KUKA KRL program: AutoChangeToolSps.src, AutoChangeToolSps.dat

--- AutoChangeToolSps.src ---
&ACCESS RV
&REL 153
&COMMENT Ansteuerung Micromaster Frequenzumrichter
&PARAM EDITMASK = *
&PARAM TEMPLATE = C:\KRC\Roboter\Template\ExpertSubmit
DEF AutoChangeToolSps(  )

;************************************************
;              CNC Robotics Ltd
;              Unit 3
;              www.cncrobotics.co.uk
;************************************************
;     Contact: helpdesk@cncrobotics.co.uk
;     Date: 05/04/24
;     Version: 1.17.54
;************************************************
; Description: sps control specific for AutoChange Tool
;************************************************


;for no tool unlock whilst spindle is running
IF (oSpindleOn) THEN    ; spindle state is true
   oToolUnlock1 = FALSE	     ; tool unlock1 state false
   oToolUnlock2 = FALSE	     ; tool unlock2 state false
ENDIF

END

--- AutoChangeToolSps.dat ---
&ACCESS  RV
&COMMENT Ansteuerung Micromaster Frequenzumrichter
&PARAM EDITMASK = *
&PARAM TEMPLATE = C:\KRC\Roboter\Template\ExpertSubmit
&REL 153
DEFDAT  AUTOCHANGETOOLSPS PUBLIC

;digital inputs
;GLOBAL SIGNAL iToolLocked $IN[] ;tool locked from spindle
;GLOBAL SIGNAL iOpenCollet $IN[] ;collet open from spindle

;digital outputs
;GLOBAL SIGNAL oToolUnlock1 $OUT[] ;Tool unlock 1
;GLOBAL SIGNAL oToolLock $OUT[] ;Tool lock for spindle
;GLOBAL SIGNAL oToolUnlock2 $OUT[] ;Tool unlock 2 to spindle



;Global Variables
GLOBAL INT nToolHeld=0 ;Current tool held by robot


ENDDAT
